FUNCTION_BLOCK DigitalInputChannel IMPLEMENTS I_DigitalInput
VAR
	input AT %I* : BOOL;
END_VAR

PROPERTY PUBLIC State : BOOL
GET
State := input;
END_GET
END_PROPERTY

END_FUNCTION_BLOCK

(* stored: Version 1.1.0.1, ProductVersion 3.1.4024.5
   POU DigitalInputChannel: Id {5c6a713e-2c69-4d9f-8dc7-efcd756feb99}, SpecialFunc None
   Property State: Id {83083960-b663-47bb-9742-2c99f61efac9}
   Get Get: Id {4ede2f07-b188-441c-a8a0-e09ad7aae6d0} *)
